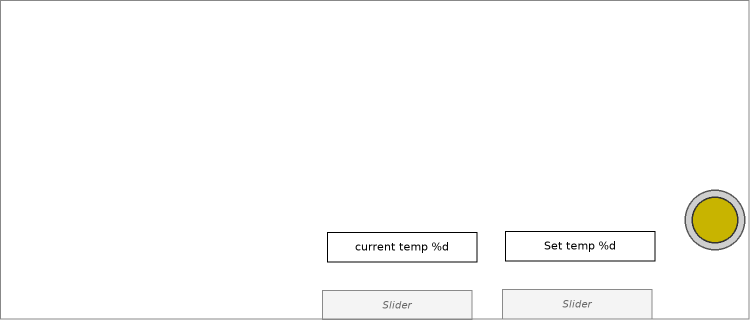
VISUALIZATION Visualization  // 750x320
    Slider (502,289 150x30), variable: MAIN.iInputsettemp, scale 0..32767
    Slider (322,290 150x30), variable: MAIN.iInputcurrenttemp, scale 0..32767
    Lamp1 (680,185 70x70), variable: MAIN.bheating, style: Lamp-Lamp1-Yellow
    Rectangle (327,232 150x30), "current temp %d", text variable: MAIN.iCurrentTemp
    Rectangle (505,231 150x30), "Set temp %d", text variable: MAIN.iSetTemp
END_VISUALIZATION

(* stored: Version 1.1.0.1, ProductVersion 3.1.4024.12
   Visu Visualization: Id {876efaee-24df-4e36-aba3-6f56e1e82840} *)
